FUNCTION_BLOCK Train1
  (* Standard: 61499-2 *)
  (* Version 0.1, 2015-00-24, Th?o, PC_THEO *)
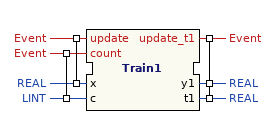
  EVENT_INPUT
    update WITH x;
    count WITH c;
  END_EVENT
  EVENT_OUTPUT
    update_t1 WITH y1, t1;
  END_EVENT
  VAR_INPUT
    x : REAL;
    c : LINT;
  END_VAR
  VAR_OUTPUT
    y1 : REAL;
    t1 : REAL;
  END_VAR
  VAR
    d : REAL;
    k : INT;
    C1y1 : REAL;
    delta : REAL;
    t : LINT := 0;
  END_VAR
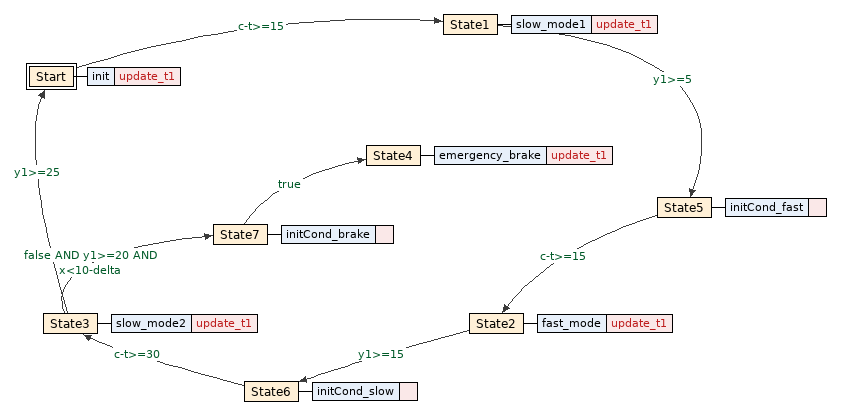
  EC_STATES
    Start : init -> update_t1;
    State1 : slow_mode1 -> update_t1;
    State2 : fast_mode -> update_t1;
    State3 : slow_mode2 -> update_t1;
    State4 : emergency_brake -> update_t1;
    State5 : initCond_fast;
    State6 : initCond_slow;
    State7 : initCond_brake;
  END_STATES
  EC_TRANSITIONS
    Start TO State1 := c-t>=15;
    State1 TO State5 := y1>=5;
    State2 TO State6 := y1>=15;
    State3 TO State7 := false AND y1>=20 AND x<10-delta;
    State3 TO Start := y1>=25;
    State5 TO State2 := c-t>=15;
    State6 TO State3 := c-t>=30;
    State7 TO State4 := true;
  END_TRANSITIONS
  ALGORITHM init IN C:
me->y1=0;
me->delta=0.0001;
me->k=1;
me->C1y1=0;
me->d=0.01;
if(me->t==0){
printf("train 1 position : %f\n", me->y1);
}
  END_ALGORITHM
  ALGORITHM slow_mode1 IN C:
//me->y1=me->d*me->k+me->C1y1;
me->y1=5;
printf("train 1 position : %f\n", me->y1);
(me->k)++;
me->t=me->c;
me->t1=me->t/(float)3;
//printf("train1 time : %d\n", me->t);
  END_ALGORITHM
  ALGORITHM fast_mode IN C:
//me->y1=2*me->d*me->k+me->C1y1;
me->y1=15;
(me->k)++;
printf("y1 : %f\n", me->y1);
me->t=me->c;
me->t1=me->t/(float)3;
//printf("train1 time : %d\n", me->t);
  END_ALGORITHM
  ALGORITHM emergency_brake IN C:
//float temp = me->y1;
float temp = 20;
//me->y1 = me->C1y1*exp(-10*me->d*me->k)+23;
me->y1 =23;
(me->k)++;


if (me->y1 - temp <= me->delta) {
	printf ("Emergency brake : Train stopped at y1 = %f and x = %f\n",me->y1, me->x);
	exit(1);
	}
  END_ALGORITHM
  ALGORITHM initCond_fast IN C:
me->k=1;
me->C1y1=me->y1;
//printf("Train 1 is going into fast mode \n");
  END_ALGORITHM
  ALGORITHM initCond_slow IN C:
me->k=1;
me->C1y1=me->y1;
//printf("Train 1 is going into slow mode \n");
  END_ALGORITHM
  ALGORITHM initCond_brake IN C:
me->k=1;
me->C1y1=me->y1-23;
printf("Emergency brake T1 !!!\n");
  END_ALGORITHM
  ALGORITHM slow_mode2 IN C:
//me->y1=me->d*me->k+me->C1y1;
me->y1=25;
printf("train 1 position : %f\n", me->y1);
(me->k)++;
me->t=me->c;
me->t1=me->t/(float)3;
//printf("train1 time : %d\n", me->t);
  END_ALGORITHM
END_FUNCTION_BLOCK
